TYPE InputBase_8311D824 :
STRUCT
END_STRUCT
END_TYPE

(* stored: Version 1.2.0.0, ProductVersion 3.1.4024.11
   DUT InputBase_8311D824: Id {6a99bae9-3c63-4a02-9ffa-7fcf72e0b93b} *)
